Fanuc KAREL source: kf00037.KL

PROGRAM KF00037
%NOLOCKGROUP
VAR
I:INTEGER;J:INTEGER;X:REAL;Y:REAL;B:BOOLEAN;C:BOOLEAN;TXT : STRING[80];TXT2 : STRING[80];AI : ARRAY[4] OF INTEGER;BI : ARRAY[4] OF INTEGER;P : XYZWPR
JP : JOINTPOS9
PF : POSITION
V1 : VECTOR
V2 : VECTOR
STATUS:INTEGER
BEGIN
--
--
--
--
--
--
--
--
--
--
AI[2]=9
I=AI[2]
END KF00037
